FUNCTION_BLOCK FB_BufferStorage
VAR_INPUT
END_VAR
VAR_OUTPUT
	{attribute 'OPC.UA.DA' := '1'}	
	localState : ST_BufferStorageState;
END_VAR
VAR
	UpperTemperatureSensor : FB_TemperatureSensor; //upper temperature sensor
	MidTemperatureSensor : FB_TemperatureSensor; //mid temperature sensor
	LowerTemperatureSensor : FB_TemperatureSensor; //lower temperature sensor
	PressureSensor : FB_PressureSensor; //pressure sensor
	stVWMZx01DefaultParameters : ST_VirtualHeatCounterDefaultParameters_Storage := (tTaskCycleTime := GlobalVariables.tTaskCycleTime_MAIN, tCtrlCycleTime := GlobalVariables.tCtrlCycleTime_MAIN);
	VWMZx01 : FB_VirtualHeatCounter_Storage := (ST_DefaultParameters := stVWMZx01DefaultParameters);
END_VAR

//sensors
UpperTemperatureSensor();
MidTemperatureSensor();
LowerTemperatureSensor();
PressureSensor();

//get sensor inputs
UpperTemperatureSensor.GetState_AI();
MidTemperatureSensor.GetState_AI();
LowerTemperatureSensor.GetState_AI();
PressureSensor.GetState_AI();

//set outputs
localState.fUpperTemperature := UpperTemperatureSensor.fTemperature;
localState.fMidTemperature := MidTemperatureSensor.fTemperature;
localState.fLowerTemperature := LowerTemperatureSensor.fTemperature;

//virtual heat counter
VWMZx01(fStorageTemperature := localState.fMidTemperature,
	fFeedTemperature := localState.fUpperTemperature,
	fReturnTemperature := localState.fLowerTemperature);

END_FUNCTION_BLOCK

(* stored: Version 1.1.0.1, ProductVersion 3.1.4024.10
   POU FB_BufferStorage: Id {2610907a-84da-47a6-a6a4-a2efbb133c01}, SpecialFunc None *)
